{attribute 'qualified_only'}
VAR_GLOBAL CONSTANT
	NumberOfMovers : UINT := 10;
	NumberOfStations : UINT := 6;
	NumberOfParts : UINT := 1;
	NumberOfTracks : UINT := 2;
END_VAR

(* stored: Version 1.1.0.1
   GVL SystemParameters: Id {a42cb835-2569-4791-97b8-892f4c778688}, ParameterList True *)
